FUNCTION F_MechToEl : LREAL
VAR_INPUT
	w_mech : LREAL;
	p : 	LREAL;
END_VAR
VAR
	w_el : LREAL;
END_VAR


w_el := w_mech * p;

IF w_el > 2*PI THEN
	w_el := w_el - 2*pi;
END_IF

F_MechToEl := w_el;

END_FUNCTION

(* stored: Version 1.1.0.1, ProductVersion 3.1.4022.17
   POU F_MechToEl: Id {5bfbe53f-56e2-49f4-b78e-8282179e9959}, SpecialFunc None *)
